TYPE ST_AxisAlarm :
STRUCT
    bError       : BOOL;
    nErrorID     : UDINT;
    eErrorSource : E_AxisErrorSource;

    bWarning     : BOOL;
    nWarningID   : UDINT;

    nRejectReason : UDINT;
END_STRUCT
END_TYPE

(* stored: Version 1.1.0.1, ProductVersion 3.1.4026.18
   DUT ST_AxisAlarm: Id {026c1a49-80b2-4404-8728-874d0f9ae498} *)
